SUBAPPLICATION Verteiler_Sitzventile (* Subapplication Type *)
  (* Standard: 61499-2 *)
  (* Version 1.0, 2023-02-11, franz *)
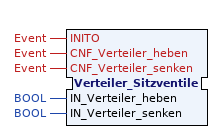
  EVENT_INPUT
    INITO;
    CNF_Verteiler_heben;
    CNF_Verteiler_senken;
  END_EVENT
  VAR_INPUT
    IN_Verteiler_heben : BOOL;
    IN_Verteiler_senken : BOOL;
  END_VAR
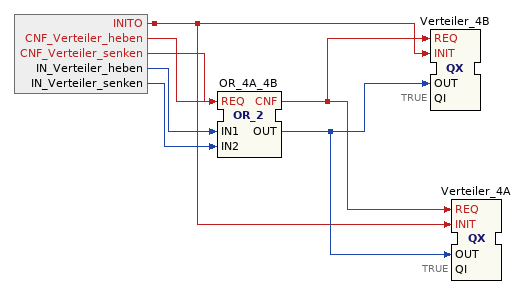
  FBS
    OR_4A_4B : OR_2; {SET_ATTRIBUTE(PinComment, IN1:Verteiler_heben)} {SET_ATTRIBUTE(PinComment, IN2:Verteiler_senken)}
    Verteiler_4B : QX(QI := TRUE);
    Verteiler_4A : QX(QI := TRUE);
  END_FBS
  EVENT_CONNECTIONS
    OR_4A_4B.CNF TO Verteiler_4B.REQ;
    OR_4A_4B.CNF TO Verteiler_4A.REQ;
    CNF_Verteiler_heben TO OR_4A_4B.REQ;
    CNF_Verteiler_senken TO OR_4A_4B.REQ;
    INITO TO Verteiler_4B.INIT;
    INITO TO Verteiler_4A.INIT;
  END_CONNECTIONS
  DATA_CONNECTIONS
    OR_4A_4B.OUT TO Verteiler_4B.OUT;
    OR_4A_4B.OUT TO Verteiler_4A.OUT;
    IN_Verteiler_heben TO OR_4A_4B.IN1;
    IN_Verteiler_senken TO OR_4A_4B.IN2;
  END_CONNECTIONS
END_SUBAPPLICATION
